PROGRAM MAIN
VAR
END_VAR

END_PROGRAM

(* stored: Version 1.1.0.1
   POU MAIN: Id {08e5a0d7-fa71-44a1-8114-bc4cc88edbfb} *)
